Fanuc KAREL source: kt00911.KL

-- PROVISIONAL review KL for V1013-1; original PC SHA256 702a6c3b5658c81308e443e4b24fbb91f6c4100a65cf747681ec7893cec3cb63
-- Incomplete behavior may be omitted. Consult companion uncertainty JSON. Do not deploy.
PROGRAM KT00911
%NOLOCKGROUP
BEGIN
  -- UNRESOLVED_PC offsets 5-31; opcodes 27,27,49,7E,AD,31,4A
  -- UNRESOLVED_PC offsets 36-40; opcodes 7F
END KT00911
